PROGRAM MAIN
VAR
  
END_VAR

HLI3_Init(); 
PRG_Messages();

(* Call CNC related code only if the HLI has been initialized succesfully! *)
IF CNCSystem.bHLIInit THEN
	PRG_CNCAxesHandler();    	
	PRG_CNCManualMode();
	PRG_CNCChannelHandler();	
	PRG_CNCVariablesViewer();	
	PRG_CNCDebug();						
END_IF
(* Reset the reset flag from HMI *)
PLCReset := FALSE;

END_PROGRAM

(* stored: Version 1.1.0.1, ProductVersion 3.1.4022.7
   POU MAIN: Id {34c8c45c-58c6-4f5f-9362-3ad98fa8450c}, SpecialFunc None *)
